FUNCTION_BLOCK EM_Tank
VAR_INPUT
	
END_VAR
VAR_OUTPUT
END_VAR
VAR
END_VAR

END_FUNCTION_BLOCK

(* stored: Version 1.1.0.1, ProductVersion 3.1.4024.13
   POU EM_Tank: Id {f3692e50-4b98-43f6-9336-6d9a3f0032b6}, SpecialFunc None *)
